// TwinCAT 3 PLC project Tc3_MC2_OOP_Library
// Title: Tc3_MC2_OOP
// Company: Unknown
// Author: Patryk Supel
// ProjectVersion: 1.0.0.0
// ProgramVersion: 3.1.4024.0
// libraries:
//   Tc2_MC2, * (Beckhoff Automation GmbH)
//   Tc2_MC2_Camming, * (Beckhoff Automation GmbH)
//   Tc2_Standard, * (Beckhoff Automation GmbH)
// project tree:
//   DUTs/Internal/ E_MotionCommand.TcDUT
//   ITFs/ itfAxisCommand.TcIO, itfCamTable.TcIO, itfCommand.TcIO, itfSynchronizedAxisCommand.TcIO
//   POUs/ Axis.TcPOU, CamTable.TcPOU
//   POUs/Internal/ AxisCommand.TcPOU, SynchronizedAxisCommand.TcPOU
//   Project Information/ F_GetCompany.TcPOU, F_GetTitle.TcPOU, F_GetVersion.TcPOU
//   Version/ Global_Version.TcGVL

// ---- DUTs/Internal/E_MotionCommand.TcDUT
//{attribute 'qualified_only'}
{attribute 'strict'}
TYPE E_MotionCommand :
(
	eNoCommand,
	ePower,
	eMoveAbsolute,
	eMoveRelative,
	eMoveVelocity,
	eHalt,
	eGearIn,
	eGearOut
);
END_TYPE

// ---- Version/Global_Version.TcGVL
{attribute 'TcGenerated'}
{attribute 'no-analysis'}
{attribute 'linkalways'}
// This function has been automatically generated from the project information.
VAR_GLOBAL CONSTANT
	{attribute 'const_non_replaced'}
	stLibVersion_Tc3_MC2_OOP : ST_LibVersion := (iMajor := 1, iMinor := 0, iBuild := 0, iRevision := 0, nFlags := 0, sVersion := '1.0.0.0');
END_VAR

// ---- ITFs/itfAxisCommand.TcIO
INTERFACE itfAxisCommand EXTENDS itfCommand

METHOD Update : MC_Error
VAR_INPUT
	Position : REAL;
	Velocity : REAL;
	EndVelocity : REAL;
	Acceleration : REAL;
	Deceleration : REAL;
	Jerk : REAL;
END_VAR
END_METHOD

END_INTERFACE

// ---- ITFs/itfCamTable.TcIO
INTERFACE itfCamTable

METHOD Select		: itfCommand
VAR_INPUT
	Periodic		: BOOL;
	MasterAbsolute	: BOOL;
	SlaveAbsolute	: BOOL;
	CamTable		: MC_CAM_REF;
END_VAR
END_METHOD

END_INTERFACE

// ---- ITFs/itfCommand.TcIO
INTERFACE itfCommand

METHOD Abort : MC_Error
VAR_INPUT
END_VAR
END_METHOD

PROPERTY Active : BOOL
GET
END_GET
END_PROPERTY

PROPERTY Busy : BOOL
GET
END_GET
END_PROPERTY

PROPERTY Command : MC_COMMAND_REF
GET
END_GET
END_PROPERTY

PROPERTY CommandAborted : BOOL
GET
END_GET
END_PROPERTY

PROPERTY Done : BOOL
GET
END_GET
END_PROPERTY

PROPERTY Error : BOOL
GET
END_GET
END_PROPERTY

PROPERTY ErrorId : UDINT
GET
END_GET
END_PROPERTY

METHOD Wait : MC_Error // This method only makes sense in the IEC 61499 environment
VAR_INPUT
	Timeout : TIME;
	AbortOnTimeout : BOOL; 
END_VAR
END_METHOD

END_INTERFACE

// ---- ITFs/itfSynchronizedAxisCommand.TcIO
INTERFACE itfSynchronizedAxisCommand EXTENDS itfAxisCommand

PROPERTY InSync : BOOL
GET
END_GET
END_PROPERTY

END_INTERFACE

// ---- POUs/Axis.TcPOU
FUNCTION_BLOCK Axis
VAR
	axisRef				: AXIS_REF;
	masterAxis			: AXIS_REF;
	motionCommand		: E_MotionCommand;
	lastMotionCommand	: E_MotionCommand;
	mcPower				: MC_Power;
	mcMoveAbsolute		: MC_MoveAbsolute;
	mcMoveRelative		: MC_MoveRelative;
	mcMoveVelocity		: MC_MoveVelocity;
	mcHalt				: MC_Halt;
	mcGearIn			: MC_GearIn;
	mcGearOut			: MC_GearOut;
END_VAR

axisRef();
//axisRef.ReadStatus();

IF lastMotionCommand <> motionCommand THEN
	
	CASE lastMotionCommand OF
		
		eNoCommand:
			;
			
		ePower:
			;
			
		eMoveAbsolute:
			mcMoveAbsolute	(Axis := THIS^.axisRef, Execute := FALSE);
			
		eMoveRelative:
			mcMoveRelative	(Axis := THIS^.axisRef, Execute := FALSE);
			
		eMoveVelocity:
			mcMoveVelocity	(Axis := THIS^.axisRef, Execute := FALSE);
			
		eHalt:
			mcHalt			(Axis := THIS^.axisRef, Execute := FALSE);
			
		eGearIn:
			mcGearIn		(Master := masterAxis, Slave := THIS^.axisRef, Execute := FALSE);
			
		eGearOut:
			mcGearOut		(Slave := THIS^.axisRef, Execute := FALSE);
			
	END_CASE
	
	lastMotionCommand := motionCommand;
	
END_IF

CASE motionCommand OF
	
	eNoCommand:
		;
		
	ePower:
		mcPower			(Axis := THIS^.axisRef);
		
	eMoveAbsolute:
		mcMoveAbsolute	(Axis := THIS^.axisRef);
		
	eMoveRelative:
		mcMoveRelative	(Axis := THIS^.axisRef);
		
	eMoveVelocity:
		mcMoveVelocity	(Axis := THIS^.axisRef);
		
	eHalt:
		mcHalt			(Axis := THIS^.axisRef);
		
	eGearIn:
		mcGearIn		(Master := masterAxis, Slave := THIS^.axisRef);
		
	eGearOut:
		mcGearOut		(Slave := THIS^.axisRef);
		
END_CASE

METHOD GearIn				: itfSynchronizedAxisCommand
VAR_INPUT
//	Execute          		: BOOL;
    RatioNumerator   		: LREAL;
    RatioDenominator 		: UINT;
//	MasterValueSource		: MC_SOURCE;
    Acceleration     		: LREAL;
    Deceleration     		: LREAL;
    Jerk             		: LREAL;
    BufferMode       		: MC_BufferMode; 
//    Options          		: ST_GearInOptions;
END_VAR
VAR_IN_OUT
	Master					: AXIS_REF;
END_VAR
VAR_INST
	gearInFb			: SynchronizedAxisCommand;
END_VAR
mcGearIn.Execute			:= TRUE;
mcGearIn.RatioNumerator		:= RatioNumerator;
mcGearIn.RatioDenominator	:= RatioDenominator;
//mcGearIn.MasterValueSource	:= MasterValueSource;
mcGearIn.Acceleration		:= Acceleration;
mcGearIn.Deceleration		:= Deceleration;
mcGearIn.Jerk				:= Jerk;
mcGearIn.BufferMode			:= BufferMode;
//mcmcGearIn.Options			:= Options;
masterAxis					:= Master;

//gearInFb._done				REF= mcGearIn.Done;
gearInFb._busy				REF= mcGearIn.Busy;
gearInFb._active			REF= mcGearIn.Active;
gearInFb._commandAborted	REF= mcGearIn.CommandAborted;
gearInFb._error				REF= mcGearIn.Error;
gearInFb._errorId			REF= mcGearIn.ErrorID;

gearInFb._inSync			REF= mcGearIn.InGear;

motionCommand := eGearIn;

GearIn := gearInFb;
END_METHOD

METHOD Halt			: itfCommand
VAR_INPUT
//	Execute      	: BOOL;
    Deceleration	: LREAL; 
    Jerk         	: LREAL;
    BufferMode   	: MC_BufferMode;
//    Options      	: ST_MoveOptions;
END_VAR
VAR_INST
	haltFb			: AxisCommand;
END_VAR
mcHalt.Execute			:= TRUE;
mcHalt.Deceleration		:= Deceleration;
mcHalt.Jerk				:= Jerk;
mcHalt.BufferMode		:= BufferMode;
//mcHalt.Options			:= Options;

haltFb._done			REF= mcHalt.Done;
haltFb._busy			REF= mcHalt.Busy;
haltFb._active			REF= mcHalt.Active;
haltFb._commandAborted	REF= mcHalt.CommandAborted;
haltFb._error			REF= mcHalt.Error;
haltFb._errorId			REF= mcHalt.ErrorID;

motionCommand := eHalt;

Halt := haltFb;
END_METHOD

METHOD MoveAbsolute : itfCommand
VAR_INPUT
//	Execute      	: BOOL;
    Position     	: LREAL; 
    Velocity     	: LREAL; 
    Acceleration 	: LREAL; 
    Deceleration 	: LREAL; 
    Jerk         	: LREAL;
    BufferMode   	: MC_BufferMode;
//    Options      	: ST_MoveOptions;
END_VAR
VAR_INST
	moveAbsoluteFb	: AxisCommand;
END_VAR
mcMoveAbsolute.Execute			:= TRUE;
mcMoveAbsolute.Position			:= Position;
mcMoveAbsolute.Velocity			:= Velocity;
mcMoveAbsolute.Acceleration		:= Acceleration;
mcMoveAbsolute.Deceleration		:= Deceleration;
mcMoveAbsolute.Jerk				:= Jerk;
mcMoveAbsolute.BufferMode		:= BufferMode;
//mcMoveAbsolute.Options			:= Options;

moveAbsoluteFb._done			REF= mcMoveAbsolute.Done;
moveAbsoluteFb._busy			REF= mcMoveAbsolute.Busy;
moveAbsoluteFb._active			REF= mcMoveAbsolute.Active;
moveAbsoluteFb._commandAborted	REF= mcMoveAbsolute.CommandAborted;
moveAbsoluteFb._error			REF= mcMoveAbsolute.Error;
moveAbsoluteFb._errorId			REF= mcMoveAbsolute.ErrorID;

motionCommand := eMoveAbsolute;

MoveAbsolute := moveAbsoluteFb;
END_METHOD

METHOD MoveRelative : itfCommand
VAR_INPUT
//	Execute      	: BOOL;
    Distance     	: LREAL; 
    Velocity     	: LREAL; 
    Acceleration 	: LREAL; 
    Deceleration 	: LREAL; 
    Jerk         	: LREAL;
    BufferMode   	: MC_BufferMode;
//    Options      	: ST_MoveOptions;
END_VAR
VAR_INST
	moveRelativeFb	: AxisCommand;
END_VAR
mcMoveRelative.Execute			:= TRUE;
mcMoveRelative.Distance			:= Distance;
mcMoveRelative.Velocity			:= Velocity;
mcMoveRelative.Acceleration		:= Acceleration;
mcMoveRelative.Deceleration		:= Deceleration;
mcMoveRelative.Jerk				:= Jerk;
mcMoveRelative.BufferMode		:= BufferMode;
//mcMoveRelative.Options			:= Options;

moveRelativeFb._done			REF= mcMoveRelative.Done;
moveRelativeFb._busy			REF= mcMoveRelative.Busy;
moveRelativeFb._active			REF= mcMoveRelative.Active;
moveRelativeFb._commandAborted	REF= mcMoveRelative.CommandAborted;
moveRelativeFb._error			REF= mcMoveRelative.Error;
moveRelativeFb._errorId			REF= mcMoveRelative.ErrorID;

motionCommand := eMoveRelative;

MoveRelative := moveRelativeFb;
END_METHOD

METHOD MoveVelocity : itfCommand
VAR_INPUT
//	Execute      	: BOOL;
    Velocity     	: LREAL; 
    Acceleration 	: LREAL; 
    Deceleration 	: LREAL; 
    Jerk         	: LREAL;
	Direction		: MC_Direction := MC_Positive_Direction;
    BufferMode   	: MC_BufferMode;
//    Options      	: ST_MoveOptions;
END_VAR
VAR_INST
	moveVelocityFb	: AxisCommand;
END_VAR
mcMoveVelocity.Execute			:= TRUE;
mcMoveVelocity.Velocity			:= Velocity;
mcMoveVelocity.Acceleration		:= Acceleration;
mcMoveVelocity.Deceleration		:= Deceleration;
mcMoveVelocity.Jerk				:= Jerk;
mcMoveVelocity.Direction		:= Direction;
mcMoveVelocity.BufferMode		:= BufferMode;
//mcMoveVelocity.Options			:= Options;

moveVelocityFb._done			REF= mcMoveVelocity.InVelocity;
moveVelocityFb._busy			REF= mcMoveVelocity.Busy;
moveVelocityFb._active			REF= mcMoveVelocity.Active;
moveVelocityFb._commandAborted	REF= mcMoveVelocity.CommandAborted;
moveVelocityFb._error			REF= mcMoveVelocity.Error;
moveVelocityFb._errorId			REF= mcMoveVelocity.ErrorID;

motionCommand := eMoveVelocity;

MoveVelocity := moveVelocityFb;
END_METHOD

METHOD Power		: itfCommand
VAR_INPUT
	Enable          : BOOL;
    Enable_Positive : BOOL;
    Enable_Negative : BOOL;
//    Override        : LREAL := 100.0;
//    BufferMode      : MC_BufferMode;
//    Options         : ST_PowerOptions;
END_VAR
VAR_INST
	powerFb			: AxisCommand;
END_VAR
mcPower.Enable			:= Enable;
mcPower.Enable_Positive	:= Enable_Positive;
mcPower.Enable_Negative	:= Enable_Negative;
//mcPower.Override		:= Override;
//mcPower.BufferMode		:= BufferMode;
//mcPower.Options			:= Options;

//powerFb._status			REF= mcPower.Status;
powerFb._busy			REF= mcPower.Busy;
powerFb._active			REF= mcPower.Active;
powerFb._error			REF= mcPower.Error;
powerFb._errorId		REF= mcPower.ErrorID;

motionCommand := ePower;

Power := powerFb;
END_METHOD

METHOD ReadStatus
VAR_INPUT
END_VAR
THIS^();
END_METHOD

METHOD Release	: UDINT
VAR_INPUT
END_VAR
;
END_METHOD

{attribute 'monitoring' := 'variable'}
PROPERTY Status : MC_AxisStates
GET
Status := axisRef.Status.MotionState;
END_GET
END_PROPERTY

END_FUNCTION_BLOCK

// ---- POUs/Internal/SynchronizedAxisCommand.TcPOU
FUNCTION_BLOCK SynchronizedAxisCommand EXTENDS AxisCommand IMPLEMENTS itfSynchronizedAxisCommand
VAR_INPUT
	_inSync	: REFERENCE TO BOOL;
END_VAR

PROPERTY InSync : BOOL
GET
InSync := _inSync;
END_GET
END_PROPERTY

END_FUNCTION_BLOCK

// ---- POUs/Internal/AxisCommand.TcPOU
FUNCTION_BLOCK AxisCommand IMPLEMENTS itfAxisCommand
VAR_INPUT
	_done			: REFERENCE TO BOOL;
	_busy			: REFERENCE TO BOOL;
	_active			: REFERENCE TO BOOL;
	_commandAborted	: REFERENCE TO BOOL;
	_error			: REFERENCE TO BOOL;
	_errorId		: REFERENCE TO UDINT;
END_VAR

{warning 'Add method implementation '}
METHOD Abort : UDINT
END_METHOD

PROPERTY Active : BOOL
GET
Active := _active;
END_GET
END_PROPERTY

PROPERTY Busy : BOOL
GET
Busy := _busy;
END_GET
END_PROPERTY

{warning 'Add property implementation'}
PROPERTY Command : MC_COMMAND_REF
GET
END_GET
END_PROPERTY

PROPERTY CommandAborted : BOOL
GET
CommandAborted := _commandAborted;
END_GET
END_PROPERTY

PROPERTY Done : BOOL
GET
Done := done;
END_GET
END_PROPERTY

PROPERTY Error : BOOL
GET
Error := _error;
END_GET
END_PROPERTY

PROPERTY ErrorId : UDINT
GET
ErrorId := _errorId;
END_GET
END_PROPERTY

{warning 'Add method implementation '}
METHOD Update		: UDINT
VAR_INPUT
	Position		: REAL;
	Velocity		: REAL;
	EndVelocity		: REAL;
	Acceleration	: REAL;
	Deceleration	: REAL;
	Jerk			: REAL;
END_VAR
END_METHOD

{warning 'Add method implementation '}
METHOD Wait			: UDINT (* This method only makes sense in the IEC 61499 environment*)
VAR_INPUT
	Timeout			: TIME;
	AbortOnTimeout	: BOOL;
END_VAR
END_METHOD

END_FUNCTION_BLOCK

// ---- POUs/CamTable.TcPOU
FUNCTION_BLOCK CamTable IMPLEMENTS itfCamTable
VAR_INPUT
END_VAR
VAR_OUTPUT
END_VAR
VAR
END_VAR

{warning 'Add method implementation '}
METHOD Select		: itfCommand
VAR_INPUT
	Periodic		: BOOL;
	MasterAbsolute	: BOOL;
	SlaveAbsolute	: BOOL;
	CamTable		: MC_CAM_REF;
END_VAR
END_METHOD

END_FUNCTION_BLOCK

// ---- Project Information/F_GetCompany.TcPOU
// This function has been automatically generated from the project information.
{attribute 'signature_flag' := '1073741824'}
{attribute 'TcGenerated'}
{attribute 'no-analysis'}
FUNCTION F_GetCompany : WSTRING
VAR_INPUT
	
END_VAR

F_GetCompany := "Unknown";

END_FUNCTION

// ---- Project Information/F_GetTitle.TcPOU
// This function has been automatically generated from the project information.
{attribute 'signature_flag' := '1073741824'}
{attribute 'TcGenerated'}
{attribute 'no-analysis'}
FUNCTION F_GetTitle : WSTRING
VAR_INPUT
	
END_VAR

F_GetTitle := "Tc3_MC2_OOP";

END_FUNCTION

// ---- Project Information/F_GetVersion.TcPOU
// This function has been automatically generated from the project information.
{attribute 'signature_flag' := '1073741824'}
{attribute 'TcGenerated'}
{attribute 'no-analysis'}
FUNCTION F_GetVersion : ST_LibVersion
VAR_INPUT
	
END_VAR

F_GetVersion.iMajor := 1;
F_GetVersion.iMinor := 0;
F_GetVersion.iBuild := 0;
F_GetVersion.iRevision := 0;
F_GetVersion.sVersion := '1.0.0.0';
F_GetVersion.nFlags := 0;

END_FUNCTION
